FUNCTION_BLOCK FB_StaticHeatingSystem
VAR_INPUT
END_VAR
VAR_OUTPUT
END_VAR
VAR
END_VAR

END_FUNCTION_BLOCK

(* stored: Version 1.1.0.1, ProductVersion 3.1.4024.10
   POU FB_StaticHeatingSystem: Id {47923f72-ad6c-4025-8311-45ce8250a43c}, SpecialFunc None *)
